// Mitsubishi GX Works2 project: z09   PLC: Q02/Q02H

PROGRAM MAIN
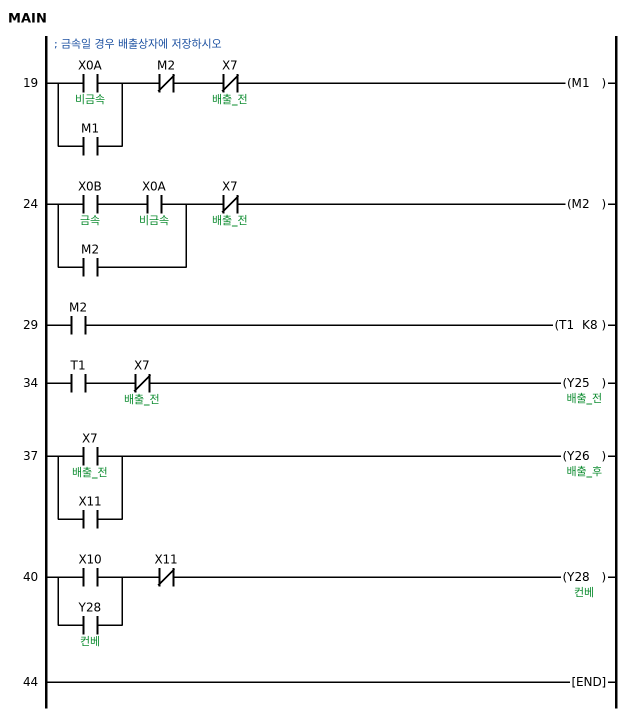
; 금속일 경우 배출상자에 저장하시오
19    LD      X0A  ; 비금속
      OR      M1
      ANI     M2
      ANI     X7  ; 배출_전
      OUT     M1
24    LD      X0B  ; 금속
      AND     X0A  ; 비금속
      OR      M2
      ANI     X7  ; 배출_전
      OUT     M2
29    LD      M2
      OUT     T1 K8
34    LD      T1
      ANI     X7  ; 배출_전
      OUT     Y25  ; 배출_전
37    LD      X7  ; 배출_전
      OR      X11
      OUT     Y26  ; 배출_후
40    LD      X10
      OR      Y28  ; 컨베
      ANI     X11
      OUT     Y28  ; 컨베
44    END
END_PROGRAM

// device comments not shown above
X0  ; 공급_후
X1  ; 공급_전
X2  ; 드릴_상
X3  ; 드릴_하
X4  ; 송출_후
X5  ; 송출_전
X6  ; 배출_후
X8  ; 매거진
X9  ; 이송감지
X0C  ; PB1
X0D  ; PB2
X0E  ; PB3
X0F  ; 비상정지
Y20  ; 공급_전
Y21  ; 공급_후
Y22  ; 드릴_실
Y23  ; 송출_전
Y24  ; 송출_후
Y27  ; 드릴_모
Y29  ; 적램
Y2A  ; 황램
Y2B  ; 녹램
